// TIA Portal V17 export
// export: Created 2025-03-10T13:11:01.0010356Z, ExportSetting WithDefaults, DisplayName Totally Integrated Automation Portal, DisplayVersion V17 Update 8, DisplayName TIA Portal Openness, DisplayVersion V17 Update 8, DisplayName TIA Portal Version Control Interface, DisplayVersion V17, DisplayName SINAMICS Startdrive Advanced, DisplayVersion V17 SP2, DisplayName SINAMICS Startdrive G110M, G120, G120C, G120D, G120P, G115D, DisplayVersion V17 SP2, DisplayName SINAMICS Startdrive G130, G150, S120, S150, SINAMICS MV, S210, DisplayVersion V17 SP2, DisplayName STEP 7 Professional, DisplayVersion V17 Update 8, DisplayName SINUMERIK ONE STEP 7 Toolbox, DisplayVersion V17 Update 12, DisplayName SINUMERIK 840D sl STEP 7 Toolbox, DisplayVersion V17 Update 12, DisplayName STEP 7 Safety, DisplayVersion V17 Update 6, DisplayName WinCC Advanced, DisplayVersion V17 Update 8
FUNCTION "FC1451_MAIN_COOLING_SYSTEM" : Void   // FC1451, LAD
{ S7_Optimized_Access := 'TRUE' }
VERSION : 0.1
// stored: AutoNumber false, IsIECCheckEnabled false, SetENOAutomatically false, UDAEnableTagReadback false
   VAR_TEMP
      COOLING_INPUT_FLOW_VALUE_NORM : Real;   // COOLING INPUT FLOW VALUE NORMALIZED
      COOLING_INPUT_FLOW_VALUE_SCALE : Real;   // COOLING INPUT FLOW VALUE SCALED
      COOLING_INPUT_FLOW_VALUE_MS : Real;   // COOLING INPUT FLOW VALUE IN M/S
      COOLING_INPUT_FLOW_VALUE_M3S : Real;   // COOLING INPUT FLOW VALUE M3/S
      COOLING_INPUT_TEMP_VALUE_AUX : Int;   // COOLING INPUT TEMPERATURE VALUE AUX
      COOLING_INPUT_TEMP_VALUE_NORM : Real;   // COOLING INPUT TEMPERATURE VALUE NORMALIZED
      COOLING_INPUT_TEMP_VALUE_SCALE : Real;   // COOLING INPUT TEMPERATURE VALUE SCALED
      COOLING_OUTPUT_FLOW_VALUE_NORM : Real;   // COOLING OUTPUT VALUE NORMALIZED
      COOLING_OUTPUT_FLOW_VALUE_SCALE : Real;   // COOLING OUTPUT VALUE SCALED
      COOLING_OUTPUT_FLOW_VALUE_MS : Real;   // COOLING OUTPUT VALUE IN M/S
      COOLING_OUTPUT_FLOW_VALUE_M3S : Real;   // COOLING OUTPUT VALUE M3/S
      COOLING_OUTPUT_TEMP_VALUE_AUX : Int;   // COOLING OUTPUT TEMPERATURE VALUE AUX
      COOLING_OUTPUT_TEMP_VALUE_NORM : Real;   // COOLING OUTPUT TEMPERATURE VALUE NORMALIZED
      COOLING_OUTPUT_TEMP_VALUE_SCALE : Real;   // COOLING OUTPUT TEMPERATURE VALUE SCALED
   END_VAR
   VAR CONSTANT
      FC_NUMBER : DInt := 1451;
   END_VAR
   VAR_TEMP   // added for the SCL form of the ladder/FBD networks
      _w1 : Bool;
   END_VAR
BEGIN

REGION Network 1: <<<<<<<<<<<<<<<<<<<< MACHINE COOLING INPUT>>>>>>>>>>>>>>>>>>>>
END_REGION

REGION Network 2: MACHINE COOLING INPUT SENSOR VALUES
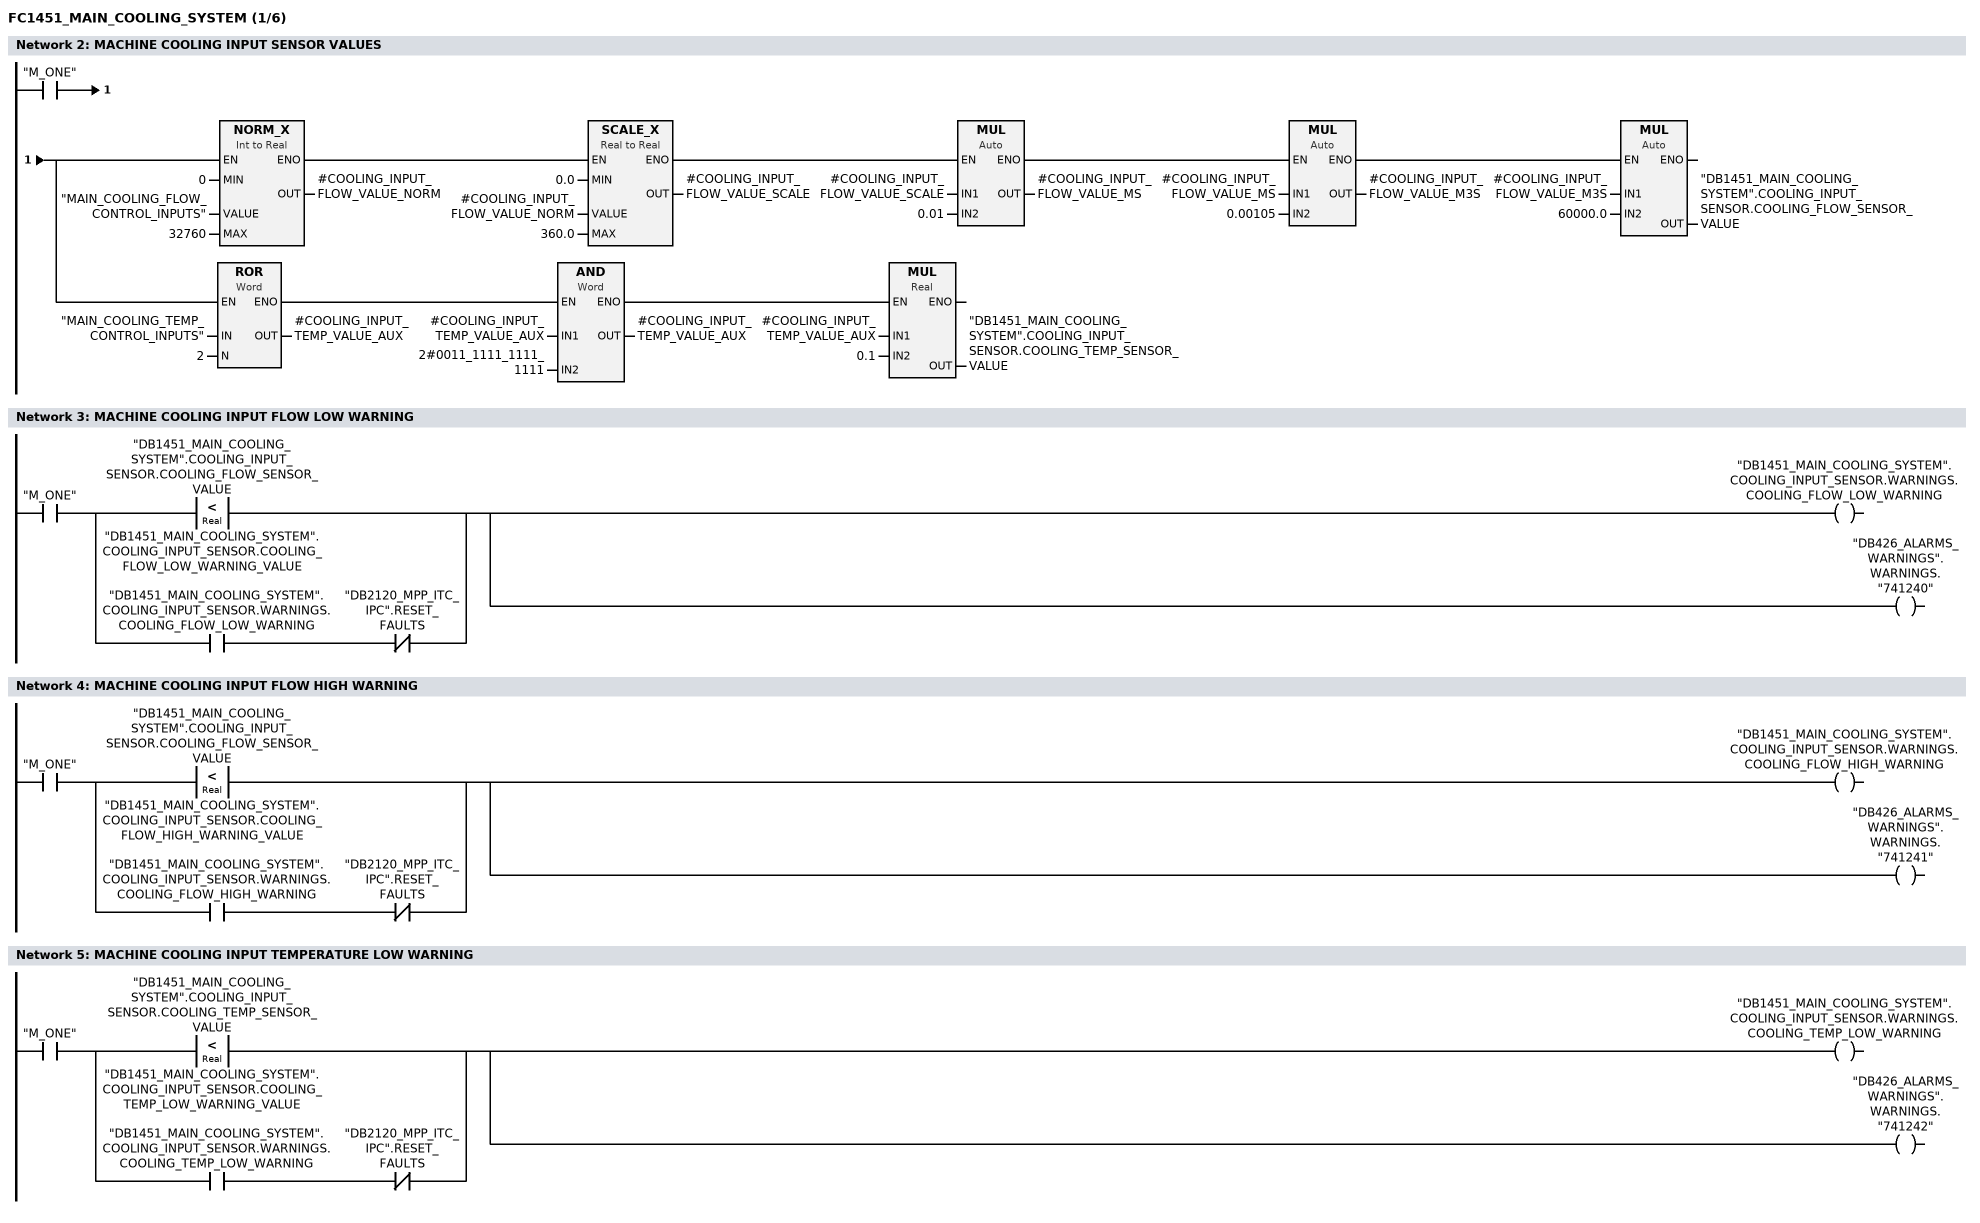
   IF "M_ONE" THEN
       #COOLING_INPUT_FLOW_VALUE_NORM := NORM_X(MIN := 0, VALUE := "MAIN_COOLING_FLOW_CONTROL_INPUTS", MAX := 32760);
       #COOLING_INPUT_FLOW_VALUE_SCALE := SCALE_X(MIN := 0.0, VALUE := #COOLING_INPUT_FLOW_VALUE_NORM, MAX := 360.0);
       #COOLING_INPUT_FLOW_VALUE_MS := #COOLING_INPUT_FLOW_VALUE_SCALE * 0.01;
       #COOLING_INPUT_FLOW_VALUE_M3S := #COOLING_INPUT_FLOW_VALUE_MS * 0.00105;
       "DB1451_MAIN_COOLING_SYSTEM".COOLING_INPUT_SENSOR.COOLING_FLOW_SENSOR_VALUE := #COOLING_INPUT_FLOW_VALUE_M3S * 60000.0;
       #COOLING_INPUT_TEMP_VALUE_AUX := ROR(IN := "MAIN_COOLING_TEMP_CONTROL_INPUTS", N := 2);
       #COOLING_INPUT_TEMP_VALUE_AUX := #COOLING_INPUT_TEMP_VALUE_AUX AND 2#0011_1111_1111_1111;
       "DB1451_MAIN_COOLING_SYSTEM".COOLING_INPUT_SENSOR.COOLING_TEMP_SENSOR_VALUE := #COOLING_INPUT_TEMP_VALUE_AUX * 0.1;
   END_IF;
END_REGION

REGION Network 3: MACHINE COOLING INPUT FLOW LOW WARNING
   RUNG wire#powerrail
      Contact( "M_ONE" )
      wire#w1
      { S7_Templates := "SrcType := Real" } LT_Contact(in1 := "DB1451_MAIN_COOLING_SYSTEM".COOLING_INPUT_SENSOR.COOLING_FLOW_SENSOR_VALUE, in2 := "DB1451_MAIN_COOLING_SYSTEM".COOLING_INPUT_SENSOR.COOLING_FLOW_LOW_WARNING_VALUE)
      wire#w2
      Coil( "DB1451_MAIN_COOLING_SYSTEM".COOLING_INPUT_SENSOR.WARNINGS.COOLING_FLOW_LOW_WARNING )
   END_RUNG
   RUNG wire#w1
      Contact( "DB1451_MAIN_COOLING_SYSTEM".COOLING_INPUT_SENSOR.WARNINGS.COOLING_FLOW_LOW_WARNING )
      I_Contact( "DB2120_MPP_ITC_IPC".RESET_FAULTS )
   END_RUNG wire#w2
   RUNG wire#w2
      Coil( "DB426_ALARMS_WARNINGS".WARNINGS."741240" )
   END_RUNG
   // the same network as SCL:
   "DB1451_MAIN_COOLING_SYSTEM".COOLING_INPUT_SENSOR.WARNINGS.COOLING_FLOW_LOW_WARNING := "M_ONE" AND (("DB1451_MAIN_COOLING_SYSTEM".COOLING_INPUT_SENSOR.COOLING_FLOW_SENSOR_VALUE < "DB1451_MAIN_COOLING_SYSTEM".COOLING_INPUT_SENSOR.COOLING_FLOW_LOW_WARNING_VALUE) OR ("DB1451_MAIN_COOLING_SYSTEM".COOLING_INPUT_SENSOR.WARNINGS.COOLING_FLOW_LOW_WARNING AND NOT "DB2120_MPP_ITC_IPC".RESET_FAULTS));
   "DB426_ALARMS_WARNINGS".WARNINGS."741240" := "DB1451_MAIN_COOLING_SYSTEM".COOLING_INPUT_SENSOR.WARNINGS.COOLING_FLOW_LOW_WARNING;
END_REGION

REGION Network 4: MACHINE COOLING INPUT FLOW HIGH WARNING
   RUNG wire#powerrail
      Contact( "M_ONE" )
      wire#w1
      { S7_Templates := "SrcType := Real" } LT_Contact(in1 := "DB1451_MAIN_COOLING_SYSTEM".COOLING_INPUT_SENSOR.COOLING_FLOW_SENSOR_VALUE, in2 := "DB1451_MAIN_COOLING_SYSTEM".COOLING_INPUT_SENSOR.COOLING_FLOW_HIGH_WARNING_VALUE)
      wire#w2
      Coil( "DB1451_MAIN_COOLING_SYSTEM".COOLING_INPUT_SENSOR.WARNINGS.COOLING_FLOW_HIGH_WARNING )
   END_RUNG
   RUNG wire#w1
      Contact( "DB1451_MAIN_COOLING_SYSTEM".COOLING_INPUT_SENSOR.WARNINGS.COOLING_FLOW_HIGH_WARNING )
      I_Contact( "DB2120_MPP_ITC_IPC".RESET_FAULTS )
   END_RUNG wire#w2
   RUNG wire#w2
      Coil( "DB426_ALARMS_WARNINGS".WARNINGS."741241" )
   END_RUNG
   // the same network as SCL:
   "DB1451_MAIN_COOLING_SYSTEM".COOLING_INPUT_SENSOR.WARNINGS.COOLING_FLOW_HIGH_WARNING := "M_ONE" AND (("DB1451_MAIN_COOLING_SYSTEM".COOLING_INPUT_SENSOR.COOLING_FLOW_SENSOR_VALUE < "DB1451_MAIN_COOLING_SYSTEM".COOLING_INPUT_SENSOR.COOLING_FLOW_HIGH_WARNING_VALUE) OR ("DB1451_MAIN_COOLING_SYSTEM".COOLING_INPUT_SENSOR.WARNINGS.COOLING_FLOW_HIGH_WARNING AND NOT "DB2120_MPP_ITC_IPC".RESET_FAULTS));
   "DB426_ALARMS_WARNINGS".WARNINGS."741241" := "DB1451_MAIN_COOLING_SYSTEM".COOLING_INPUT_SENSOR.WARNINGS.COOLING_FLOW_HIGH_WARNING;
END_REGION

REGION Network 5: MACHINE COOLING INPUT TEMPERATURE LOW WARNING
   RUNG wire#powerrail
      Contact( "M_ONE" )
      wire#w1
      { S7_Templates := "SrcType := Real" } LT_Contact(in1 := "DB1451_MAIN_COOLING_SYSTEM".COOLING_INPUT_SENSOR.COOLING_TEMP_SENSOR_VALUE, in2 := "DB1451_MAIN_COOLING_SYSTEM".COOLING_INPUT_SENSOR.COOLING_TEMP_LOW_WARNING_VALUE)
      wire#w2
      Coil( "DB1451_MAIN_COOLING_SYSTEM".COOLING_INPUT_SENSOR.WARNINGS.COOLING_TEMP_LOW_WARNING )
   END_RUNG
   RUNG wire#w1
      Contact( "DB1451_MAIN_COOLING_SYSTEM".COOLING_INPUT_SENSOR.WARNINGS.COOLING_TEMP_LOW_WARNING )
      I_Contact( "DB2120_MPP_ITC_IPC".RESET_FAULTS )
   END_RUNG wire#w2
   RUNG wire#w2
      Coil( "DB426_ALARMS_WARNINGS".WARNINGS."741242" )
   END_RUNG
   // the same network as SCL:
   "DB1451_MAIN_COOLING_SYSTEM".COOLING_INPUT_SENSOR.WARNINGS.COOLING_TEMP_LOW_WARNING := "M_ONE" AND (("DB1451_MAIN_COOLING_SYSTEM".COOLING_INPUT_SENSOR.COOLING_TEMP_SENSOR_VALUE < "DB1451_MAIN_COOLING_SYSTEM".COOLING_INPUT_SENSOR.COOLING_TEMP_LOW_WARNING_VALUE) OR ("DB1451_MAIN_COOLING_SYSTEM".COOLING_INPUT_SENSOR.WARNINGS.COOLING_TEMP_LOW_WARNING AND NOT "DB2120_MPP_ITC_IPC".RESET_FAULTS));
   "DB426_ALARMS_WARNINGS".WARNINGS."741242" := "DB1451_MAIN_COOLING_SYSTEM".COOLING_INPUT_SENSOR.WARNINGS.COOLING_TEMP_LOW_WARNING;
END_REGION

REGION Network 6: MACHINE COOLING INPUT TEMPERATURE HIGH WARNINGS
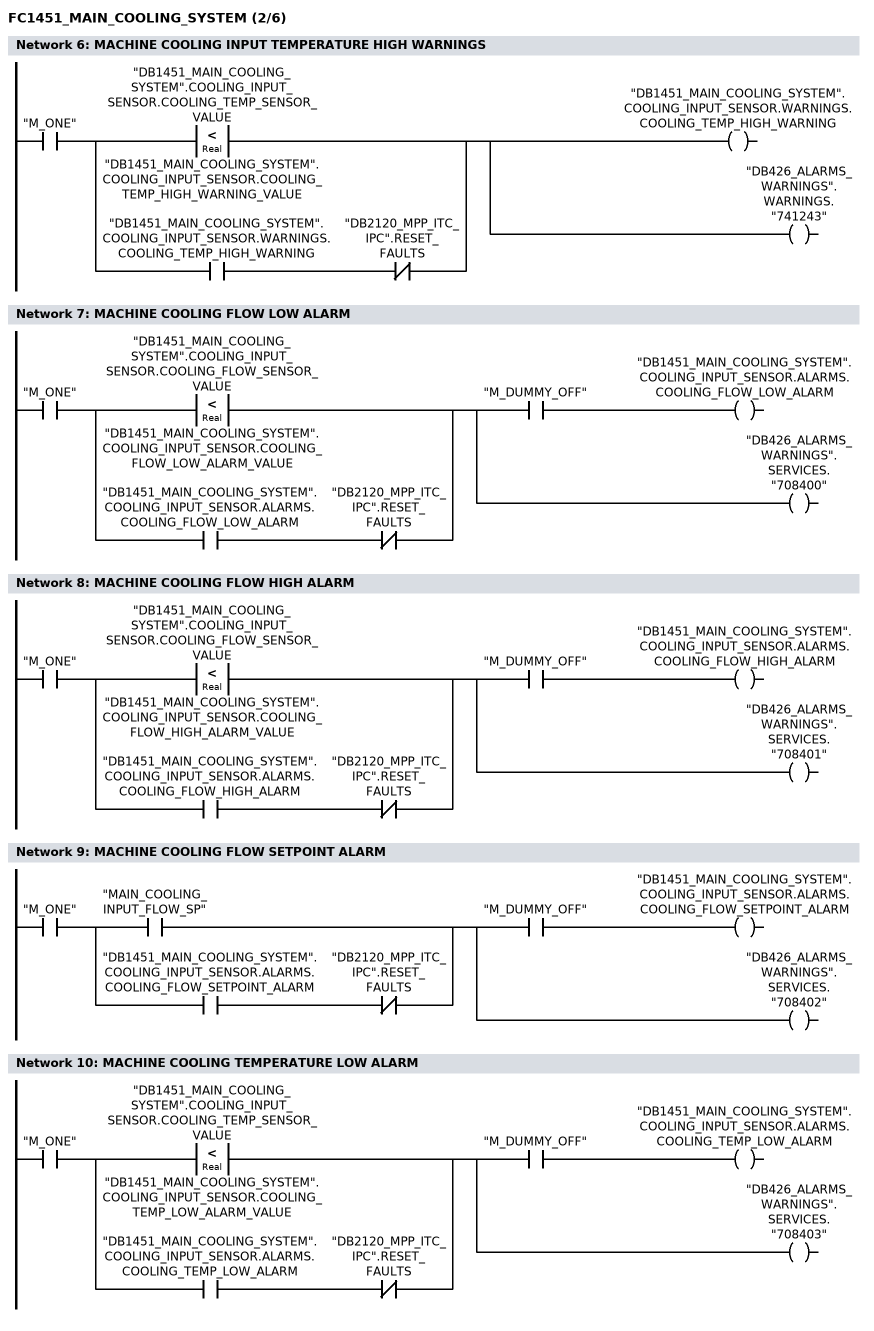
   RUNG wire#powerrail
      Contact( "M_ONE" )
      wire#w1
      { S7_Templates := "SrcType := Real" } LT_Contact(in1 := "DB1451_MAIN_COOLING_SYSTEM".COOLING_INPUT_SENSOR.COOLING_TEMP_SENSOR_VALUE, in2 := "DB1451_MAIN_COOLING_SYSTEM".COOLING_INPUT_SENSOR.COOLING_TEMP_HIGH_WARNING_VALUE)
      wire#w2
      Coil( "DB1451_MAIN_COOLING_SYSTEM".COOLING_INPUT_SENSOR.WARNINGS.COOLING_TEMP_HIGH_WARNING )
   END_RUNG
   RUNG wire#w1
      Contact( "DB1451_MAIN_COOLING_SYSTEM".COOLING_INPUT_SENSOR.WARNINGS.COOLING_TEMP_HIGH_WARNING )
      I_Contact( "DB2120_MPP_ITC_IPC".RESET_FAULTS )
   END_RUNG wire#w2
   RUNG wire#w2
      Coil( "DB426_ALARMS_WARNINGS".WARNINGS."741243" )
   END_RUNG
   // the same network as SCL:
   "DB1451_MAIN_COOLING_SYSTEM".COOLING_INPUT_SENSOR.WARNINGS.COOLING_TEMP_HIGH_WARNING := "M_ONE" AND (("DB1451_MAIN_COOLING_SYSTEM".COOLING_INPUT_SENSOR.COOLING_TEMP_SENSOR_VALUE < "DB1451_MAIN_COOLING_SYSTEM".COOLING_INPUT_SENSOR.COOLING_TEMP_HIGH_WARNING_VALUE) OR ("DB1451_MAIN_COOLING_SYSTEM".COOLING_INPUT_SENSOR.WARNINGS.COOLING_TEMP_HIGH_WARNING AND NOT "DB2120_MPP_ITC_IPC".RESET_FAULTS));
   "DB426_ALARMS_WARNINGS".WARNINGS."741243" := "DB1451_MAIN_COOLING_SYSTEM".COOLING_INPUT_SENSOR.WARNINGS.COOLING_TEMP_HIGH_WARNING;
END_REGION

REGION Network 7: MACHINE COOLING FLOW LOW ALARM
   RUNG wire#powerrail
      Contact( "M_ONE" )
      wire#w1
      { S7_Templates := "SrcType := Real" } LT_Contact(in1 := "DB1451_MAIN_COOLING_SYSTEM".COOLING_INPUT_SENSOR.COOLING_FLOW_SENSOR_VALUE, in2 := "DB1451_MAIN_COOLING_SYSTEM".COOLING_INPUT_SENSOR.COOLING_FLOW_LOW_ALARM_VALUE)
      wire#w2
      Contact( "M_DUMMY_OFF" )
      Coil( "DB1451_MAIN_COOLING_SYSTEM".COOLING_INPUT_SENSOR.ALARMS.COOLING_FLOW_LOW_ALARM )
   END_RUNG
   RUNG wire#w1
      Contact( "DB1451_MAIN_COOLING_SYSTEM".COOLING_INPUT_SENSOR.ALARMS.COOLING_FLOW_LOW_ALARM )
      I_Contact( "DB2120_MPP_ITC_IPC".RESET_FAULTS )
   END_RUNG wire#w2
   RUNG wire#w2
      Coil( "DB426_ALARMS_WARNINGS".SERVICES."708400" )
   END_RUNG
   // the same network as SCL:
   #_w1 := "M_ONE" AND (("DB1451_MAIN_COOLING_SYSTEM".COOLING_INPUT_SENSOR.COOLING_FLOW_SENSOR_VALUE < "DB1451_MAIN_COOLING_SYSTEM".COOLING_INPUT_SENSOR.COOLING_FLOW_LOW_ALARM_VALUE) OR ("DB1451_MAIN_COOLING_SYSTEM".COOLING_INPUT_SENSOR.ALARMS.COOLING_FLOW_LOW_ALARM AND NOT "DB2120_MPP_ITC_IPC".RESET_FAULTS));
   "DB1451_MAIN_COOLING_SYSTEM".COOLING_INPUT_SENSOR.ALARMS.COOLING_FLOW_LOW_ALARM := #_w1 AND "M_DUMMY_OFF";
   "DB426_ALARMS_WARNINGS".SERVICES."708400" := #_w1;
END_REGION

REGION Network 8: MACHINE COOLING FLOW HIGH ALARM
   RUNG wire#powerrail
      Contact( "M_ONE" )
      wire#w1
      { S7_Templates := "SrcType := Real" } LT_Contact(in1 := "DB1451_MAIN_COOLING_SYSTEM".COOLING_INPUT_SENSOR.COOLING_FLOW_SENSOR_VALUE, in2 := "DB1451_MAIN_COOLING_SYSTEM".COOLING_INPUT_SENSOR.COOLING_FLOW_HIGH_ALARM_VALUE)
      wire#w2
      Contact( "M_DUMMY_OFF" )
      Coil( "DB1451_MAIN_COOLING_SYSTEM".COOLING_INPUT_SENSOR.ALARMS.COOLING_FLOW_HIGH_ALARM )
   END_RUNG
   RUNG wire#w1
      Contact( "DB1451_MAIN_COOLING_SYSTEM".COOLING_INPUT_SENSOR.ALARMS.COOLING_FLOW_HIGH_ALARM )
      I_Contact( "DB2120_MPP_ITC_IPC".RESET_FAULTS )
   END_RUNG wire#w2
   RUNG wire#w2
      Coil( "DB426_ALARMS_WARNINGS".SERVICES."708401" )
   END_RUNG
   // the same network as SCL:
   #_w1 := "M_ONE" AND (("DB1451_MAIN_COOLING_SYSTEM".COOLING_INPUT_SENSOR.COOLING_FLOW_SENSOR_VALUE < "DB1451_MAIN_COOLING_SYSTEM".COOLING_INPUT_SENSOR.COOLING_FLOW_HIGH_ALARM_VALUE) OR ("DB1451_MAIN_COOLING_SYSTEM".COOLING_INPUT_SENSOR.ALARMS.COOLING_FLOW_HIGH_ALARM AND NOT "DB2120_MPP_ITC_IPC".RESET_FAULTS));
   "DB1451_MAIN_COOLING_SYSTEM".COOLING_INPUT_SENSOR.ALARMS.COOLING_FLOW_HIGH_ALARM := #_w1 AND "M_DUMMY_OFF";
   "DB426_ALARMS_WARNINGS".SERVICES."708401" := #_w1;
END_REGION

REGION Network 9: MACHINE COOLING FLOW SETPOINT ALARM
   RUNG wire#powerrail
      Contact( "M_ONE" )
      wire#w1
      Contact( "MAIN_COOLING_INPUT_FLOW_SP" )
      wire#w2
      Contact( "M_DUMMY_OFF" )
      Coil( "DB1451_MAIN_COOLING_SYSTEM".COOLING_INPUT_SENSOR.ALARMS.COOLING_FLOW_SETPOINT_ALARM )
   END_RUNG
   RUNG wire#w1
      Contact( "DB1451_MAIN_COOLING_SYSTEM".COOLING_INPUT_SENSOR.ALARMS.COOLING_FLOW_SETPOINT_ALARM )
      I_Contact( "DB2120_MPP_ITC_IPC".RESET_FAULTS )
   END_RUNG wire#w2
   RUNG wire#w2
      Coil( "DB426_ALARMS_WARNINGS".SERVICES."708402" )
   END_RUNG
   // the same network as SCL:
   #_w1 := "M_ONE" AND ("MAIN_COOLING_INPUT_FLOW_SP" OR ("DB1451_MAIN_COOLING_SYSTEM".COOLING_INPUT_SENSOR.ALARMS.COOLING_FLOW_SETPOINT_ALARM AND NOT "DB2120_MPP_ITC_IPC".RESET_FAULTS));
   "DB1451_MAIN_COOLING_SYSTEM".COOLING_INPUT_SENSOR.ALARMS.COOLING_FLOW_SETPOINT_ALARM := #_w1 AND "M_DUMMY_OFF";
   "DB426_ALARMS_WARNINGS".SERVICES."708402" := #_w1;
END_REGION

REGION Network 10: MACHINE COOLING TEMPERATURE LOW ALARM
   RUNG wire#powerrail
      Contact( "M_ONE" )
      wire#w1
      { S7_Templates := "SrcType := Real" } LT_Contact(in1 := "DB1451_MAIN_COOLING_SYSTEM".COOLING_INPUT_SENSOR.COOLING_TEMP_SENSOR_VALUE, in2 := "DB1451_MAIN_COOLING_SYSTEM".COOLING_INPUT_SENSOR.COOLING_TEMP_LOW_ALARM_VALUE)
      wire#w2
      Contact( "M_DUMMY_OFF" )
      Coil( "DB1451_MAIN_COOLING_SYSTEM".COOLING_INPUT_SENSOR.ALARMS.COOLING_TEMP_LOW_ALARM )
   END_RUNG
   RUNG wire#w1
      Contact( "DB1451_MAIN_COOLING_SYSTEM".COOLING_INPUT_SENSOR.ALARMS.COOLING_TEMP_LOW_ALARM )
      I_Contact( "DB2120_MPP_ITC_IPC".RESET_FAULTS )
   END_RUNG wire#w2
   RUNG wire#w2
      Coil( "DB426_ALARMS_WARNINGS".SERVICES."708403" )
   END_RUNG
   // the same network as SCL:
   #_w1 := "M_ONE" AND (("DB1451_MAIN_COOLING_SYSTEM".COOLING_INPUT_SENSOR.COOLING_TEMP_SENSOR_VALUE < "DB1451_MAIN_COOLING_SYSTEM".COOLING_INPUT_SENSOR.COOLING_TEMP_LOW_ALARM_VALUE) OR ("DB1451_MAIN_COOLING_SYSTEM".COOLING_INPUT_SENSOR.ALARMS.COOLING_TEMP_LOW_ALARM AND NOT "DB2120_MPP_ITC_IPC".RESET_FAULTS));
   "DB1451_MAIN_COOLING_SYSTEM".COOLING_INPUT_SENSOR.ALARMS.COOLING_TEMP_LOW_ALARM := #_w1 AND "M_DUMMY_OFF";
   "DB426_ALARMS_WARNINGS".SERVICES."708403" := #_w1;
END_REGION

REGION Network 11: MACHINE COOLING TEMPERATURE HIGH ALARM
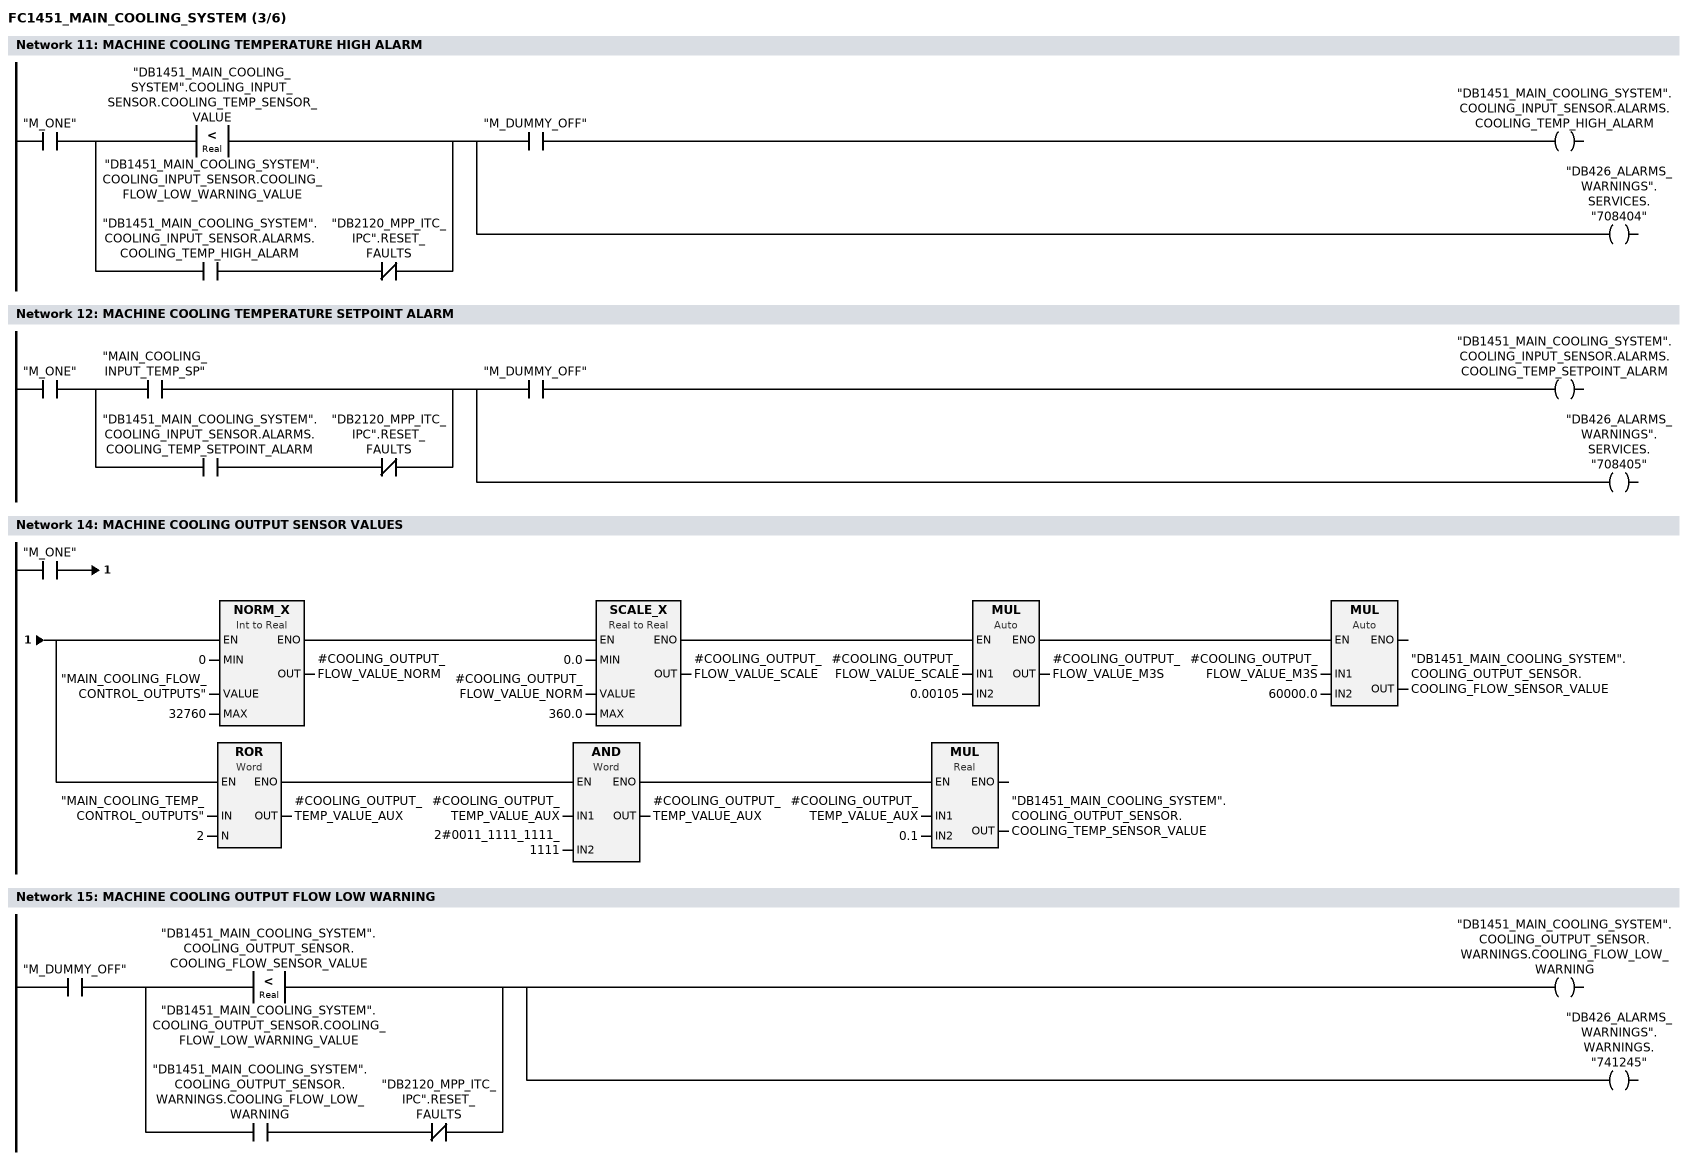
   RUNG wire#powerrail
      Contact( "M_ONE" )
      wire#w1
      { S7_Templates := "SrcType := Real" } LT_Contact(in1 := "DB1451_MAIN_COOLING_SYSTEM".COOLING_INPUT_SENSOR.COOLING_TEMP_SENSOR_VALUE, in2 := "DB1451_MAIN_COOLING_SYSTEM".COOLING_INPUT_SENSOR.COOLING_FLOW_LOW_WARNING_VALUE)
      wire#w2
      Contact( "M_DUMMY_OFF" )
      Coil( "DB1451_MAIN_COOLING_SYSTEM".COOLING_INPUT_SENSOR.ALARMS.COOLING_TEMP_HIGH_ALARM )
   END_RUNG
   RUNG wire#w1
      Contact( "DB1451_MAIN_COOLING_SYSTEM".COOLING_INPUT_SENSOR.ALARMS.COOLING_TEMP_HIGH_ALARM )
      I_Contact( "DB2120_MPP_ITC_IPC".RESET_FAULTS )
   END_RUNG wire#w2
   RUNG wire#w2
      Coil( "DB426_ALARMS_WARNINGS".SERVICES."708404" )
   END_RUNG
   // the same network as SCL:
   #_w1 := "M_ONE" AND (("DB1451_MAIN_COOLING_SYSTEM".COOLING_INPUT_SENSOR.COOLING_TEMP_SENSOR_VALUE < "DB1451_MAIN_COOLING_SYSTEM".COOLING_INPUT_SENSOR.COOLING_FLOW_LOW_WARNING_VALUE) OR ("DB1451_MAIN_COOLING_SYSTEM".COOLING_INPUT_SENSOR.ALARMS.COOLING_TEMP_HIGH_ALARM AND NOT "DB2120_MPP_ITC_IPC".RESET_FAULTS));
   "DB1451_MAIN_COOLING_SYSTEM".COOLING_INPUT_SENSOR.ALARMS.COOLING_TEMP_HIGH_ALARM := #_w1 AND "M_DUMMY_OFF";
   "DB426_ALARMS_WARNINGS".SERVICES."708404" := #_w1;
END_REGION

REGION Network 12: MACHINE COOLING TEMPERATURE SETPOINT ALARM
   RUNG wire#powerrail
      Contact( "M_ONE" )
      wire#w1
      Contact( "MAIN_COOLING_INPUT_TEMP_SP" )
      wire#w2
      Contact( "M_DUMMY_OFF" )
      Coil( "DB1451_MAIN_COOLING_SYSTEM".COOLING_INPUT_SENSOR.ALARMS.COOLING_TEMP_SETPOINT_ALARM )
   END_RUNG
   RUNG wire#w1
      Contact( "DB1451_MAIN_COOLING_SYSTEM".COOLING_INPUT_SENSOR.ALARMS.COOLING_TEMP_SETPOINT_ALARM )
      I_Contact( "DB2120_MPP_ITC_IPC".RESET_FAULTS )
   END_RUNG wire#w2
   RUNG wire#w2
      Coil( "DB426_ALARMS_WARNINGS".SERVICES."708405" )
   END_RUNG
   // the same network as SCL:
   #_w1 := "M_ONE" AND ("MAIN_COOLING_INPUT_TEMP_SP" OR ("DB1451_MAIN_COOLING_SYSTEM".COOLING_INPUT_SENSOR.ALARMS.COOLING_TEMP_SETPOINT_ALARM AND NOT "DB2120_MPP_ITC_IPC".RESET_FAULTS));
   "DB1451_MAIN_COOLING_SYSTEM".COOLING_INPUT_SENSOR.ALARMS.COOLING_TEMP_SETPOINT_ALARM := #_w1 AND "M_DUMMY_OFF";
   "DB426_ALARMS_WARNINGS".SERVICES."708405" := #_w1;
END_REGION

REGION Network 13: <<<<<<<<<<<<<<<<<<<< MACHINE COOLING OUTPUT>>>>>>>>>>>>>>>>>>>>
END_REGION

REGION Network 14: MACHINE COOLING OUTPUT SENSOR VALUES
   IF "M_ONE" THEN
       #COOLING_OUTPUT_FLOW_VALUE_NORM := NORM_X(MIN := 0, VALUE := "MAIN_COOLING_FLOW_CONTROL_OUTPUTS", MAX := 32760);
       #COOLING_OUTPUT_FLOW_VALUE_SCALE := SCALE_X(MIN := 0.0, VALUE := #COOLING_OUTPUT_FLOW_VALUE_NORM, MAX := 360.0);
       #COOLING_OUTPUT_FLOW_VALUE_M3S := #COOLING_OUTPUT_FLOW_VALUE_SCALE * 0.00105;
       "DB1451_MAIN_COOLING_SYSTEM".COOLING_OUTPUT_SENSOR.COOLING_FLOW_SENSOR_VALUE := #COOLING_OUTPUT_FLOW_VALUE_M3S * 60000.0;
       #COOLING_OUTPUT_TEMP_VALUE_AUX := ROR(IN := "MAIN_COOLING_TEMP_CONTROL_OUTPUTS", N := 2);
       #COOLING_OUTPUT_TEMP_VALUE_AUX := #COOLING_OUTPUT_TEMP_VALUE_AUX AND 2#0011_1111_1111_1111;
       "DB1451_MAIN_COOLING_SYSTEM".COOLING_OUTPUT_SENSOR.COOLING_TEMP_SENSOR_VALUE := #COOLING_OUTPUT_TEMP_VALUE_AUX * 0.1;
   END_IF;
END_REGION

REGION Network 15: MACHINE COOLING OUTPUT FLOW LOW WARNING
   RUNG wire#powerrail
      Contact( "M_DUMMY_OFF" )
      wire#w1
      { S7_Templates := "SrcType := Real" } LT_Contact(in1 := "DB1451_MAIN_COOLING_SYSTEM".COOLING_OUTPUT_SENSOR.COOLING_FLOW_SENSOR_VALUE, in2 := "DB1451_MAIN_COOLING_SYSTEM".COOLING_OUTPUT_SENSOR.COOLING_FLOW_LOW_WARNING_VALUE)
      wire#w2
      Coil( "DB1451_MAIN_COOLING_SYSTEM".COOLING_OUTPUT_SENSOR.WARNINGS.COOLING_FLOW_LOW_WARNING )
   END_RUNG
   RUNG wire#w1
      Contact( "DB1451_MAIN_COOLING_SYSTEM".COOLING_OUTPUT_SENSOR.WARNINGS.COOLING_FLOW_LOW_WARNING )
      I_Contact( "DB2120_MPP_ITC_IPC".RESET_FAULTS )
   END_RUNG wire#w2
   RUNG wire#w2
      Coil( "DB426_ALARMS_WARNINGS".WARNINGS."741245" )
   END_RUNG
   // the same network as SCL:
   "DB1451_MAIN_COOLING_SYSTEM".COOLING_OUTPUT_SENSOR.WARNINGS.COOLING_FLOW_LOW_WARNING := "M_DUMMY_OFF" AND (("DB1451_MAIN_COOLING_SYSTEM".COOLING_OUTPUT_SENSOR.COOLING_FLOW_SENSOR_VALUE < "DB1451_MAIN_COOLING_SYSTEM".COOLING_OUTPUT_SENSOR.COOLING_FLOW_LOW_WARNING_VALUE) OR ("DB1451_MAIN_COOLING_SYSTEM".COOLING_OUTPUT_SENSOR.WARNINGS.COOLING_FLOW_LOW_WARNING AND NOT "DB2120_MPP_ITC_IPC".RESET_FAULTS));
   "DB426_ALARMS_WARNINGS".WARNINGS."741245" := "DB1451_MAIN_COOLING_SYSTEM".COOLING_OUTPUT_SENSOR.WARNINGS.COOLING_FLOW_LOW_WARNING;
END_REGION

REGION Network 16: MACHINE COOLING OUTPUT FLOW HIGH WARNING
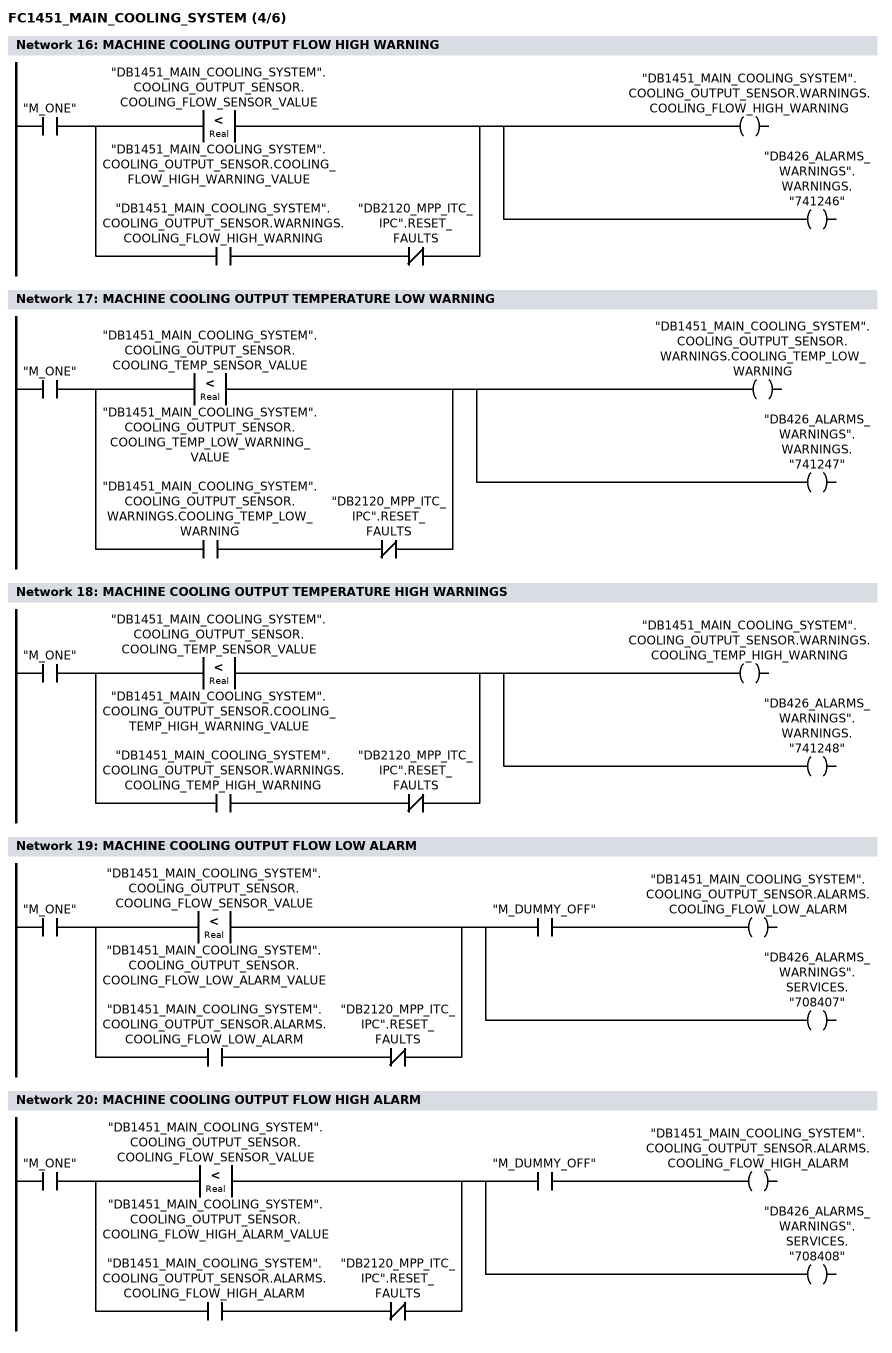
   RUNG wire#powerrail
      Contact( "M_ONE" )
      wire#w1
      { S7_Templates := "SrcType := Real" } LT_Contact(in1 := "DB1451_MAIN_COOLING_SYSTEM".COOLING_OUTPUT_SENSOR.COOLING_FLOW_SENSOR_VALUE, in2 := "DB1451_MAIN_COOLING_SYSTEM".COOLING_OUTPUT_SENSOR.COOLING_FLOW_HIGH_WARNING_VALUE)
      wire#w2
      Coil( "DB1451_MAIN_COOLING_SYSTEM".COOLING_OUTPUT_SENSOR.WARNINGS.COOLING_FLOW_HIGH_WARNING )
   END_RUNG
   RUNG wire#w1
      Contact( "DB1451_MAIN_COOLING_SYSTEM".COOLING_OUTPUT_SENSOR.WARNINGS.COOLING_FLOW_HIGH_WARNING )
      I_Contact( "DB2120_MPP_ITC_IPC".RESET_FAULTS )
   END_RUNG wire#w2
   RUNG wire#w2
      Coil( "DB426_ALARMS_WARNINGS".WARNINGS."741246" )
   END_RUNG
   // the same network as SCL:
   "DB1451_MAIN_COOLING_SYSTEM".COOLING_OUTPUT_SENSOR.WARNINGS.COOLING_FLOW_HIGH_WARNING := "M_ONE" AND (("DB1451_MAIN_COOLING_SYSTEM".COOLING_OUTPUT_SENSOR.COOLING_FLOW_SENSOR_VALUE < "DB1451_MAIN_COOLING_SYSTEM".COOLING_OUTPUT_SENSOR.COOLING_FLOW_HIGH_WARNING_VALUE) OR ("DB1451_MAIN_COOLING_SYSTEM".COOLING_OUTPUT_SENSOR.WARNINGS.COOLING_FLOW_HIGH_WARNING AND NOT "DB2120_MPP_ITC_IPC".RESET_FAULTS));
   "DB426_ALARMS_WARNINGS".WARNINGS."741246" := "DB1451_MAIN_COOLING_SYSTEM".COOLING_OUTPUT_SENSOR.WARNINGS.COOLING_FLOW_HIGH_WARNING;
END_REGION

REGION Network 17: MACHINE COOLING OUTPUT TEMPERATURE LOW WARNING
   RUNG wire#powerrail
      Contact( "M_ONE" )
      wire#w1
      { S7_Templates := "SrcType := Real" } LT_Contact(in1 := "DB1451_MAIN_COOLING_SYSTEM".COOLING_OUTPUT_SENSOR.COOLING_TEMP_SENSOR_VALUE, in2 := "DB1451_MAIN_COOLING_SYSTEM".COOLING_OUTPUT_SENSOR.COOLING_TEMP_LOW_WARNING_VALUE)
      wire#w2
      Coil( "DB1451_MAIN_COOLING_SYSTEM".COOLING_OUTPUT_SENSOR.WARNINGS.COOLING_TEMP_LOW_WARNING )
   END_RUNG
   RUNG wire#w1
      Contact( "DB1451_MAIN_COOLING_SYSTEM".COOLING_OUTPUT_SENSOR.WARNINGS.COOLING_TEMP_LOW_WARNING )
      I_Contact( "DB2120_MPP_ITC_IPC".RESET_FAULTS )
   END_RUNG wire#w2
   RUNG wire#w2
      Coil( "DB426_ALARMS_WARNINGS".WARNINGS."741247" )
   END_RUNG
   // the same network as SCL:
   "DB1451_MAIN_COOLING_SYSTEM".COOLING_OUTPUT_SENSOR.WARNINGS.COOLING_TEMP_LOW_WARNING := "M_ONE" AND (("DB1451_MAIN_COOLING_SYSTEM".COOLING_OUTPUT_SENSOR.COOLING_TEMP_SENSOR_VALUE < "DB1451_MAIN_COOLING_SYSTEM".COOLING_OUTPUT_SENSOR.COOLING_TEMP_LOW_WARNING_VALUE) OR ("DB1451_MAIN_COOLING_SYSTEM".COOLING_OUTPUT_SENSOR.WARNINGS.COOLING_TEMP_LOW_WARNING AND NOT "DB2120_MPP_ITC_IPC".RESET_FAULTS));
   "DB426_ALARMS_WARNINGS".WARNINGS."741247" := "DB1451_MAIN_COOLING_SYSTEM".COOLING_OUTPUT_SENSOR.WARNINGS.COOLING_TEMP_LOW_WARNING;
END_REGION

REGION Network 18: MACHINE COOLING OUTPUT TEMPERATURE HIGH WARNINGS
   RUNG wire#powerrail
      Contact( "M_ONE" )
      wire#w1
      { S7_Templates := "SrcType := Real" } LT_Contact(in1 := "DB1451_MAIN_COOLING_SYSTEM".COOLING_OUTPUT_SENSOR.COOLING_TEMP_SENSOR_VALUE, in2 := "DB1451_MAIN_COOLING_SYSTEM".COOLING_OUTPUT_SENSOR.COOLING_TEMP_HIGH_WARNING_VALUE)
      wire#w2
      Coil( "DB1451_MAIN_COOLING_SYSTEM".COOLING_OUTPUT_SENSOR.WARNINGS.COOLING_TEMP_HIGH_WARNING )
   END_RUNG
   RUNG wire#w1
      Contact( "DB1451_MAIN_COOLING_SYSTEM".COOLING_OUTPUT_SENSOR.WARNINGS.COOLING_TEMP_HIGH_WARNING )
      I_Contact( "DB2120_MPP_ITC_IPC".RESET_FAULTS )
   END_RUNG wire#w2
   RUNG wire#w2
      Coil( "DB426_ALARMS_WARNINGS".WARNINGS."741248" )
   END_RUNG
   // the same network as SCL:
   "DB1451_MAIN_COOLING_SYSTEM".COOLING_OUTPUT_SENSOR.WARNINGS.COOLING_TEMP_HIGH_WARNING := "M_ONE" AND (("DB1451_MAIN_COOLING_SYSTEM".COOLING_OUTPUT_SENSOR.COOLING_TEMP_SENSOR_VALUE < "DB1451_MAIN_COOLING_SYSTEM".COOLING_OUTPUT_SENSOR.COOLING_TEMP_HIGH_WARNING_VALUE) OR ("DB1451_MAIN_COOLING_SYSTEM".COOLING_OUTPUT_SENSOR.WARNINGS.COOLING_TEMP_HIGH_WARNING AND NOT "DB2120_MPP_ITC_IPC".RESET_FAULTS));
   "DB426_ALARMS_WARNINGS".WARNINGS."741248" := "DB1451_MAIN_COOLING_SYSTEM".COOLING_OUTPUT_SENSOR.WARNINGS.COOLING_TEMP_HIGH_WARNING;
END_REGION

REGION Network 19: MACHINE COOLING OUTPUT FLOW LOW ALARM
   RUNG wire#powerrail
      Contact( "M_ONE" )
      wire#w1
      { S7_Templates := "SrcType := Real" } LT_Contact(in1 := "DB1451_MAIN_COOLING_SYSTEM".COOLING_OUTPUT_SENSOR.COOLING_FLOW_SENSOR_VALUE, in2 := "DB1451_MAIN_COOLING_SYSTEM".COOLING_OUTPUT_SENSOR.COOLING_FLOW_LOW_ALARM_VALUE)
      wire#w2
      Contact( "M_DUMMY_OFF" )
      Coil( "DB1451_MAIN_COOLING_SYSTEM".COOLING_OUTPUT_SENSOR.ALARMS.COOLING_FLOW_LOW_ALARM )
   END_RUNG
   RUNG wire#w1
      Contact( "DB1451_MAIN_COOLING_SYSTEM".COOLING_OUTPUT_SENSOR.ALARMS.COOLING_FLOW_LOW_ALARM )
      I_Contact( "DB2120_MPP_ITC_IPC".RESET_FAULTS )
   END_RUNG wire#w2
   RUNG wire#w2
      Coil( "DB426_ALARMS_WARNINGS".SERVICES."708407" )
   END_RUNG
   // the same network as SCL:
   #_w1 := "M_ONE" AND (("DB1451_MAIN_COOLING_SYSTEM".COOLING_OUTPUT_SENSOR.COOLING_FLOW_SENSOR_VALUE < "DB1451_MAIN_COOLING_SYSTEM".COOLING_OUTPUT_SENSOR.COOLING_FLOW_LOW_ALARM_VALUE) OR ("DB1451_MAIN_COOLING_SYSTEM".COOLING_OUTPUT_SENSOR.ALARMS.COOLING_FLOW_LOW_ALARM AND NOT "DB2120_MPP_ITC_IPC".RESET_FAULTS));
   "DB1451_MAIN_COOLING_SYSTEM".COOLING_OUTPUT_SENSOR.ALARMS.COOLING_FLOW_LOW_ALARM := #_w1 AND "M_DUMMY_OFF";
   "DB426_ALARMS_WARNINGS".SERVICES."708407" := #_w1;
END_REGION

REGION Network 20: MACHINE COOLING OUTPUT FLOW HIGH ALARM
   RUNG wire#powerrail
      Contact( "M_ONE" )
      wire#w1
      { S7_Templates := "SrcType := Real" } LT_Contact(in1 := "DB1451_MAIN_COOLING_SYSTEM".COOLING_OUTPUT_SENSOR.COOLING_FLOW_SENSOR_VALUE, in2 := "DB1451_MAIN_COOLING_SYSTEM".COOLING_OUTPUT_SENSOR.COOLING_FLOW_HIGH_ALARM_VALUE)
      wire#w2
      Contact( "M_DUMMY_OFF" )
      Coil( "DB1451_MAIN_COOLING_SYSTEM".COOLING_OUTPUT_SENSOR.ALARMS.COOLING_FLOW_HIGH_ALARM )
   END_RUNG
   RUNG wire#w1
      Contact( "DB1451_MAIN_COOLING_SYSTEM".COOLING_OUTPUT_SENSOR.ALARMS.COOLING_FLOW_HIGH_ALARM )
      I_Contact( "DB2120_MPP_ITC_IPC".RESET_FAULTS )
   END_RUNG wire#w2
   RUNG wire#w2
      Coil( "DB426_ALARMS_WARNINGS".SERVICES."708408" )
   END_RUNG
   // the same network as SCL:
   #_w1 := "M_ONE" AND (("DB1451_MAIN_COOLING_SYSTEM".COOLING_OUTPUT_SENSOR.COOLING_FLOW_SENSOR_VALUE < "DB1451_MAIN_COOLING_SYSTEM".COOLING_OUTPUT_SENSOR.COOLING_FLOW_HIGH_ALARM_VALUE) OR ("DB1451_MAIN_COOLING_SYSTEM".COOLING_OUTPUT_SENSOR.ALARMS.COOLING_FLOW_HIGH_ALARM AND NOT "DB2120_MPP_ITC_IPC".RESET_FAULTS));
   "DB1451_MAIN_COOLING_SYSTEM".COOLING_OUTPUT_SENSOR.ALARMS.COOLING_FLOW_HIGH_ALARM := #_w1 AND "M_DUMMY_OFF";
   "DB426_ALARMS_WARNINGS".SERVICES."708408" := #_w1;
END_REGION

REGION Network 21: MACHINE COOLING OUTPUT FLOW SETPOINT ALARM
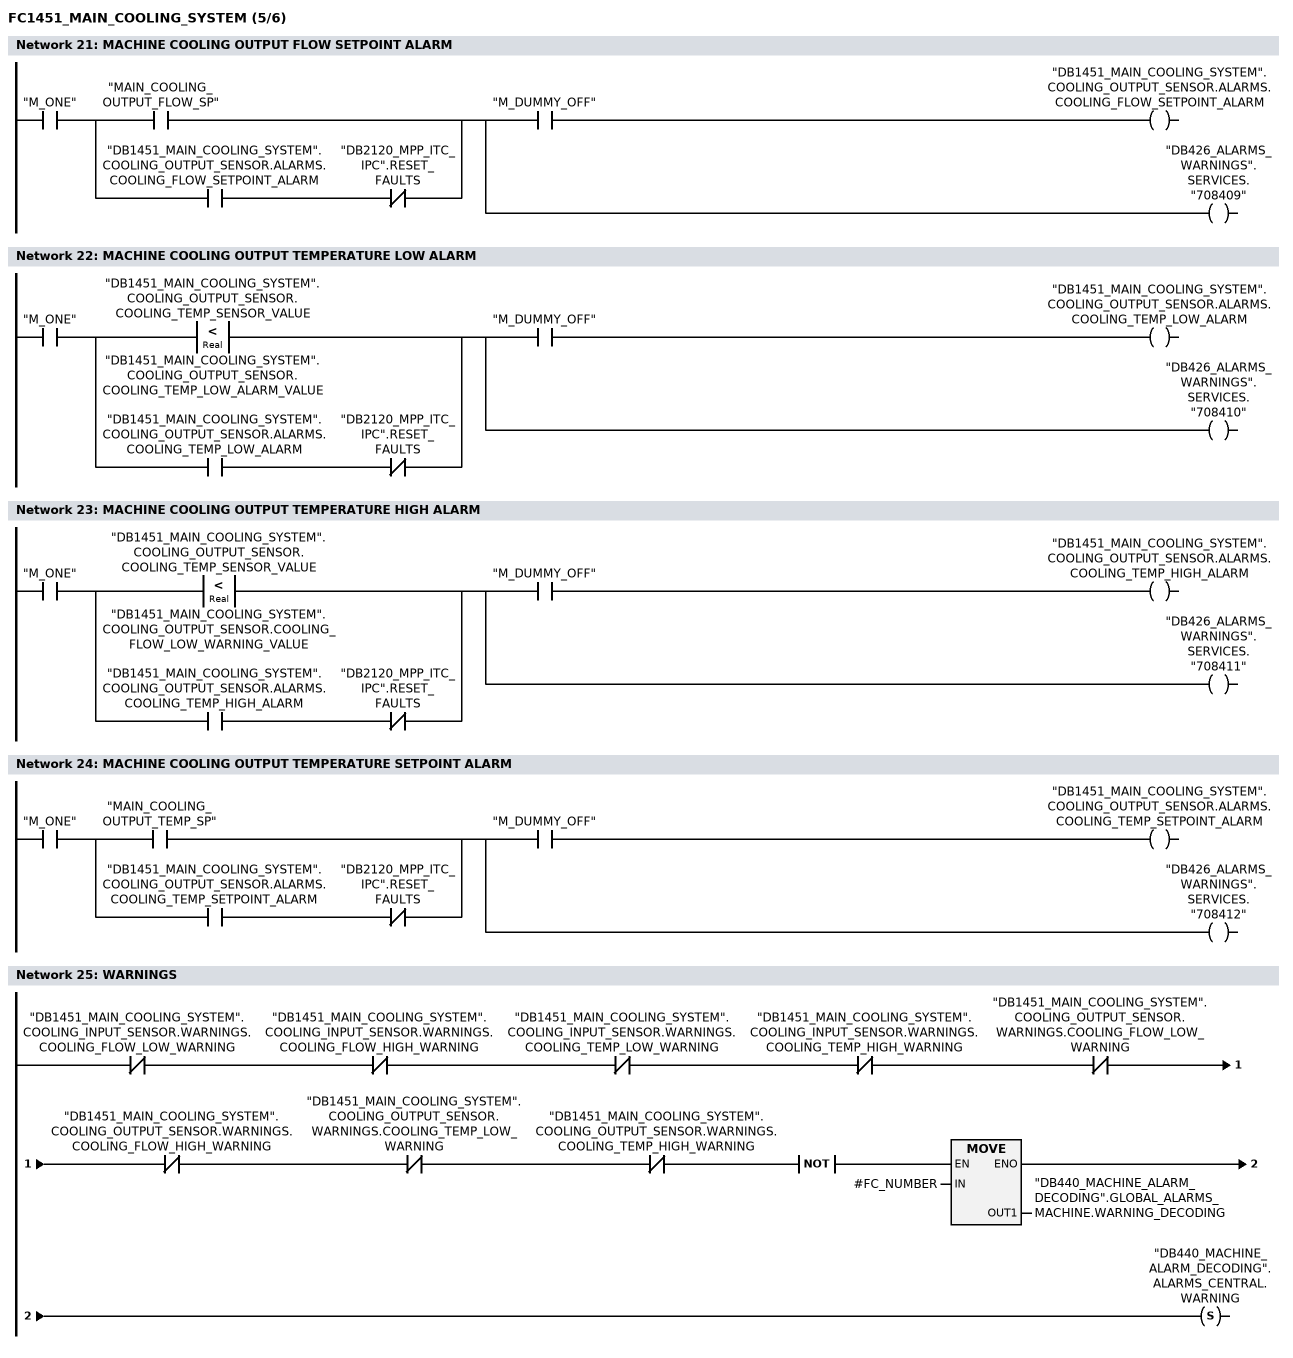
   RUNG wire#powerrail
      Contact( "M_ONE" )
      wire#w1
      Contact( "MAIN_COOLING_OUTPUT_FLOW_SP" )
      wire#w2
      Contact( "M_DUMMY_OFF" )
      Coil( "DB1451_MAIN_COOLING_SYSTEM".COOLING_OUTPUT_SENSOR.ALARMS.COOLING_FLOW_SETPOINT_ALARM )
   END_RUNG
   RUNG wire#w1
      Contact( "DB1451_MAIN_COOLING_SYSTEM".COOLING_OUTPUT_SENSOR.ALARMS.COOLING_FLOW_SETPOINT_ALARM )
      I_Contact( "DB2120_MPP_ITC_IPC".RESET_FAULTS )
   END_RUNG wire#w2
   RUNG wire#w2
      Coil( "DB426_ALARMS_WARNINGS".SERVICES."708409" )
   END_RUNG
   // the same network as SCL:
   #_w1 := "M_ONE" AND ("MAIN_COOLING_OUTPUT_FLOW_SP" OR ("DB1451_MAIN_COOLING_SYSTEM".COOLING_OUTPUT_SENSOR.ALARMS.COOLING_FLOW_SETPOINT_ALARM AND NOT "DB2120_MPP_ITC_IPC".RESET_FAULTS));
   "DB1451_MAIN_COOLING_SYSTEM".COOLING_OUTPUT_SENSOR.ALARMS.COOLING_FLOW_SETPOINT_ALARM := #_w1 AND "M_DUMMY_OFF";
   "DB426_ALARMS_WARNINGS".SERVICES."708409" := #_w1;
END_REGION

REGION Network 22: MACHINE COOLING OUTPUT TEMPERATURE LOW ALARM
   RUNG wire#powerrail
      Contact( "M_ONE" )
      wire#w1
      { S7_Templates := "SrcType := Real" } LT_Contact(in1 := "DB1451_MAIN_COOLING_SYSTEM".COOLING_OUTPUT_SENSOR.COOLING_TEMP_SENSOR_VALUE, in2 := "DB1451_MAIN_COOLING_SYSTEM".COOLING_OUTPUT_SENSOR.COOLING_TEMP_LOW_ALARM_VALUE)
      wire#w2
      Contact( "M_DUMMY_OFF" )
      Coil( "DB1451_MAIN_COOLING_SYSTEM".COOLING_OUTPUT_SENSOR.ALARMS.COOLING_TEMP_LOW_ALARM )
   END_RUNG
   RUNG wire#w1
      Contact( "DB1451_MAIN_COOLING_SYSTEM".COOLING_OUTPUT_SENSOR.ALARMS.COOLING_TEMP_LOW_ALARM )
      I_Contact( "DB2120_MPP_ITC_IPC".RESET_FAULTS )
   END_RUNG wire#w2
   RUNG wire#w2
      Coil( "DB426_ALARMS_WARNINGS".SERVICES."708410" )
   END_RUNG
   // the same network as SCL:
   #_w1 := "M_ONE" AND (("DB1451_MAIN_COOLING_SYSTEM".COOLING_OUTPUT_SENSOR.COOLING_TEMP_SENSOR_VALUE < "DB1451_MAIN_COOLING_SYSTEM".COOLING_OUTPUT_SENSOR.COOLING_TEMP_LOW_ALARM_VALUE) OR ("DB1451_MAIN_COOLING_SYSTEM".COOLING_OUTPUT_SENSOR.ALARMS.COOLING_TEMP_LOW_ALARM AND NOT "DB2120_MPP_ITC_IPC".RESET_FAULTS));
   "DB1451_MAIN_COOLING_SYSTEM".COOLING_OUTPUT_SENSOR.ALARMS.COOLING_TEMP_LOW_ALARM := #_w1 AND "M_DUMMY_OFF";
   "DB426_ALARMS_WARNINGS".SERVICES."708410" := #_w1;
END_REGION

REGION Network 23: MACHINE COOLING OUTPUT TEMPERATURE HIGH ALARM
   RUNG wire#powerrail
      Contact( "M_ONE" )
      wire#w1
      { S7_Templates := "SrcType := Real" } LT_Contact(in1 := "DB1451_MAIN_COOLING_SYSTEM".COOLING_OUTPUT_SENSOR.COOLING_TEMP_SENSOR_VALUE, in2 := "DB1451_MAIN_COOLING_SYSTEM".COOLING_OUTPUT_SENSOR.COOLING_FLOW_LOW_WARNING_VALUE)
      wire#w2
      Contact( "M_DUMMY_OFF" )
      Coil( "DB1451_MAIN_COOLING_SYSTEM".COOLING_OUTPUT_SENSOR.ALARMS.COOLING_TEMP_HIGH_ALARM )
   END_RUNG
   RUNG wire#w1
      Contact( "DB1451_MAIN_COOLING_SYSTEM".COOLING_OUTPUT_SENSOR.ALARMS.COOLING_TEMP_HIGH_ALARM )
      I_Contact( "DB2120_MPP_ITC_IPC".RESET_FAULTS )
   END_RUNG wire#w2
   RUNG wire#w2
      Coil( "DB426_ALARMS_WARNINGS".SERVICES."708411" )
   END_RUNG
   // the same network as SCL:
   #_w1 := "M_ONE" AND (("DB1451_MAIN_COOLING_SYSTEM".COOLING_OUTPUT_SENSOR.COOLING_TEMP_SENSOR_VALUE < "DB1451_MAIN_COOLING_SYSTEM".COOLING_OUTPUT_SENSOR.COOLING_FLOW_LOW_WARNING_VALUE) OR ("DB1451_MAIN_COOLING_SYSTEM".COOLING_OUTPUT_SENSOR.ALARMS.COOLING_TEMP_HIGH_ALARM AND NOT "DB2120_MPP_ITC_IPC".RESET_FAULTS));
   "DB1451_MAIN_COOLING_SYSTEM".COOLING_OUTPUT_SENSOR.ALARMS.COOLING_TEMP_HIGH_ALARM := #_w1 AND "M_DUMMY_OFF";
   "DB426_ALARMS_WARNINGS".SERVICES."708411" := #_w1;
END_REGION

REGION Network 24: MACHINE COOLING OUTPUT TEMPERATURE SETPOINT ALARM
   RUNG wire#powerrail
      Contact( "M_ONE" )
      wire#w1
      Contact( "MAIN_COOLING_OUTPUT_TEMP_SP" )
      wire#w2
      Contact( "M_DUMMY_OFF" )
      Coil( "DB1451_MAIN_COOLING_SYSTEM".COOLING_OUTPUT_SENSOR.ALARMS.COOLING_TEMP_SETPOINT_ALARM )
   END_RUNG
   RUNG wire#w1
      Contact( "DB1451_MAIN_COOLING_SYSTEM".COOLING_OUTPUT_SENSOR.ALARMS.COOLING_TEMP_SETPOINT_ALARM )
      I_Contact( "DB2120_MPP_ITC_IPC".RESET_FAULTS )
   END_RUNG wire#w2
   RUNG wire#w2
      Coil( "DB426_ALARMS_WARNINGS".SERVICES."708412" )
   END_RUNG
   // the same network as SCL:
   #_w1 := "M_ONE" AND ("MAIN_COOLING_OUTPUT_TEMP_SP" OR ("DB1451_MAIN_COOLING_SYSTEM".COOLING_OUTPUT_SENSOR.ALARMS.COOLING_TEMP_SETPOINT_ALARM AND NOT "DB2120_MPP_ITC_IPC".RESET_FAULTS));
   "DB1451_MAIN_COOLING_SYSTEM".COOLING_OUTPUT_SENSOR.ALARMS.COOLING_TEMP_SETPOINT_ALARM := #_w1 AND "M_DUMMY_OFF";
   "DB426_ALARMS_WARNINGS".SERVICES."708412" := #_w1;
END_REGION

REGION Network 25: WARNINGS
   RUNG wire#powerrail
      I_Contact( "DB1451_MAIN_COOLING_SYSTEM".COOLING_INPUT_SENSOR.WARNINGS.COOLING_FLOW_LOW_WARNING )
      I_Contact( "DB1451_MAIN_COOLING_SYSTEM".COOLING_INPUT_SENSOR.WARNINGS.COOLING_FLOW_HIGH_WARNING )
      I_Contact( "DB1451_MAIN_COOLING_SYSTEM".COOLING_INPUT_SENSOR.WARNINGS.COOLING_TEMP_LOW_WARNING )
      I_Contact( "DB1451_MAIN_COOLING_SYSTEM".COOLING_INPUT_SENSOR.WARNINGS.COOLING_TEMP_HIGH_WARNING )
      I_Contact( "DB1451_MAIN_COOLING_SYSTEM".COOLING_OUTPUT_SENSOR.WARNINGS.COOLING_FLOW_LOW_WARNING )
      I_Contact( "DB1451_MAIN_COOLING_SYSTEM".COOLING_OUTPUT_SENSOR.WARNINGS.COOLING_FLOW_HIGH_WARNING )
      I_Contact( "DB1451_MAIN_COOLING_SYSTEM".COOLING_OUTPUT_SENSOR.WARNINGS.COOLING_TEMP_LOW_WARNING )
      I_Contact( "DB1451_MAIN_COOLING_SYSTEM".COOLING_OUTPUT_SENSOR.WARNINGS.COOLING_TEMP_HIGH_WARNING )
      Not()
      Move(in := #FC_NUMBER, out1 => "DB440_MACHINE_ALARM_DECODING".GLOBAL_ALARMS_MACHINE.WARNING_DECODING)
      S_Coil( "DB440_MACHINE_ALARM_DECODING".ALARMS_CENTRAL.WARNING )
   END_RUNG
   // the same network as SCL:
   IF NOT (NOT "DB1451_MAIN_COOLING_SYSTEM".COOLING_INPUT_SENSOR.WARNINGS.COOLING_FLOW_LOW_WARNING AND NOT "DB1451_MAIN_COOLING_SYSTEM".COOLING_INPUT_SENSOR.WARNINGS.COOLING_FLOW_HIGH_WARNING AND NOT "DB1451_MAIN_COOLING_SYSTEM".COOLING_INPUT_SENSOR.WARNINGS.COOLING_TEMP_LOW_WARNING AND NOT "DB1451_MAIN_COOLING_SYSTEM".COOLING_INPUT_SENSOR.WARNINGS.COOLING_TEMP_HIGH_WARNING AND NOT "DB1451_MAIN_COOLING_SYSTEM".COOLING_OUTPUT_SENSOR.WARNINGS.COOLING_FLOW_LOW_WARNING AND NOT "DB1451_MAIN_COOLING_SYSTEM".COOLING_OUTPUT_SENSOR.WARNINGS.COOLING_FLOW_HIGH_WARNING AND NOT "DB1451_MAIN_COOLING_SYSTEM".COOLING_OUTPUT_SENSOR.WARNINGS.COOLING_TEMP_LOW_WARNING AND NOT "DB1451_MAIN_COOLING_SYSTEM".COOLING_OUTPUT_SENSOR.WARNINGS.COOLING_TEMP_HIGH_WARNING) THEN
       "DB440_MACHINE_ALARM_DECODING".GLOBAL_ALARMS_MACHINE.WARNING_DECODING := #FC_NUMBER;
       "DB440_MACHINE_ALARM_DECODING".ALARMS_CENTRAL.WARNING := TRUE;
   END_IF;
END_REGION

REGION Network 26: INMEDIATE STOP ALARMS
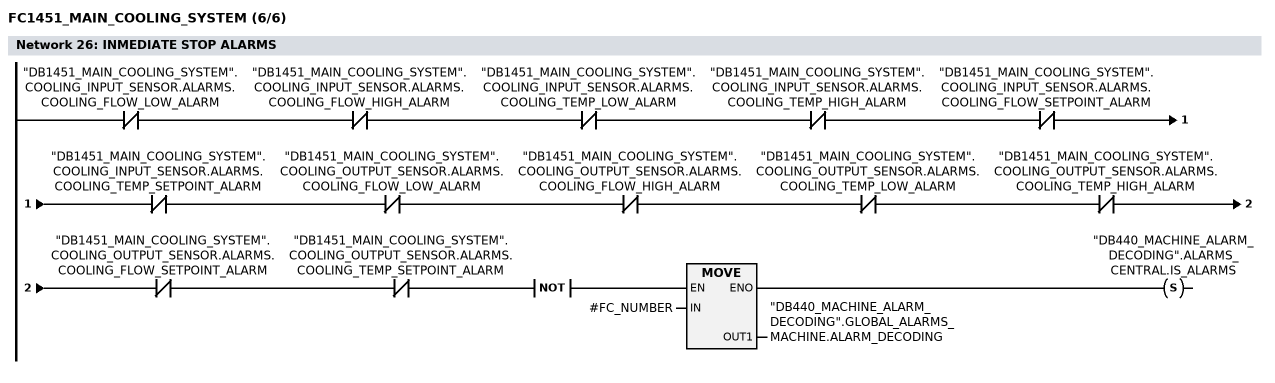
   RUNG wire#powerrail
      I_Contact( "DB1451_MAIN_COOLING_SYSTEM".COOLING_INPUT_SENSOR.ALARMS.COOLING_FLOW_LOW_ALARM )
      I_Contact( "DB1451_MAIN_COOLING_SYSTEM".COOLING_INPUT_SENSOR.ALARMS.COOLING_FLOW_HIGH_ALARM )
      I_Contact( "DB1451_MAIN_COOLING_SYSTEM".COOLING_INPUT_SENSOR.ALARMS.COOLING_TEMP_LOW_ALARM )
      I_Contact( "DB1451_MAIN_COOLING_SYSTEM".COOLING_INPUT_SENSOR.ALARMS.COOLING_TEMP_HIGH_ALARM )
      I_Contact( "DB1451_MAIN_COOLING_SYSTEM".COOLING_INPUT_SENSOR.ALARMS.COOLING_FLOW_SETPOINT_ALARM )
      I_Contact( "DB1451_MAIN_COOLING_SYSTEM".COOLING_INPUT_SENSOR.ALARMS.COOLING_TEMP_SETPOINT_ALARM )
      I_Contact( "DB1451_MAIN_COOLING_SYSTEM".COOLING_OUTPUT_SENSOR.ALARMS.COOLING_FLOW_LOW_ALARM )
      I_Contact( "DB1451_MAIN_COOLING_SYSTEM".COOLING_OUTPUT_SENSOR.ALARMS.COOLING_FLOW_HIGH_ALARM )
      I_Contact( "DB1451_MAIN_COOLING_SYSTEM".COOLING_OUTPUT_SENSOR.ALARMS.COOLING_TEMP_LOW_ALARM )
      I_Contact( "DB1451_MAIN_COOLING_SYSTEM".COOLING_OUTPUT_SENSOR.ALARMS.COOLING_TEMP_HIGH_ALARM )
      I_Contact( "DB1451_MAIN_COOLING_SYSTEM".COOLING_OUTPUT_SENSOR.ALARMS.COOLING_FLOW_SETPOINT_ALARM )
      I_Contact( "DB1451_MAIN_COOLING_SYSTEM".COOLING_OUTPUT_SENSOR.ALARMS.COOLING_TEMP_SETPOINT_ALARM )
      Not()
      Move(in := #FC_NUMBER, out1 => "DB440_MACHINE_ALARM_DECODING".GLOBAL_ALARMS_MACHINE.ALARM_DECODING)
      S_Coil( "DB440_MACHINE_ALARM_DECODING".ALARMS_CENTRAL.IS_ALARMS )
   END_RUNG
   // the same network as SCL:
   IF NOT (NOT "DB1451_MAIN_COOLING_SYSTEM".COOLING_INPUT_SENSOR.ALARMS.COOLING_FLOW_LOW_ALARM AND NOT "DB1451_MAIN_COOLING_SYSTEM".COOLING_INPUT_SENSOR.ALARMS.COOLING_FLOW_HIGH_ALARM AND NOT "DB1451_MAIN_COOLING_SYSTEM".COOLING_INPUT_SENSOR.ALARMS.COOLING_TEMP_LOW_ALARM AND NOT "DB1451_MAIN_COOLING_SYSTEM".COOLING_INPUT_SENSOR.ALARMS.COOLING_TEMP_HIGH_ALARM AND NOT "DB1451_MAIN_COOLING_SYSTEM".COOLING_INPUT_SENSOR.ALARMS.COOLING_FLOW_SETPOINT_ALARM AND NOT "DB1451_MAIN_COOLING_SYSTEM".COOLING_INPUT_SENSOR.ALARMS.COOLING_TEMP_SETPOINT_ALARM AND NOT "DB1451_MAIN_COOLING_SYSTEM".COOLING_OUTPUT_SENSOR.ALARMS.COOLING_FLOW_LOW_ALARM AND NOT "DB1451_MAIN_COOLING_SYSTEM".COOLING_OUTPUT_SENSOR.ALARMS.COOLING_FLOW_HIGH_ALARM AND NOT "DB1451_MAIN_COOLING_SYSTEM".COOLING_OUTPUT_SENSOR.ALARMS.COOLING_TEMP_LOW_ALARM AND NOT "DB1451_MAIN_COOLING_SYSTEM".COOLING_OUTPUT_SENSOR.ALARMS.COOLING_TEMP_HIGH_ALARM AND NOT "DB1451_MAIN_COOLING_SYSTEM".COOLING_OUTPUT_SENSOR.ALARMS.COOLING_FLOW_SETPOINT_ALARM AND NOT "DB1451_MAIN_COOLING_SYSTEM".COOLING_OUTPUT_SENSOR.ALARMS.COOLING_TEMP_SETPOINT_ALARM) THEN
       "DB440_MACHINE_ALARM_DECODING".GLOBAL_ALARMS_MACHINE.ALARM_DECODING := #FC_NUMBER;
       "DB440_MACHINE_ALARM_DECODING".ALARMS_CENTRAL.IS_ALARMS := TRUE;
   END_IF;
END_REGION
END_FUNCTION
